// TIA Portal V20 export
DATA_BLOCK "Simulation_DB"   // DB105
// stored: InstanceOfName Unit1.Em4.Simulation, InstanceOfType FB, Namespace Unit1.Em4
"Unit1.Em4.Simulation"
   // VAR
   //    Simulation_addon_Instance { S7_SetPoint := 'True'} : "Simulation_addon";
   // END_VAR
BEGIN
END_DATA_BLOCK
